VISUALIZATION VISU_Home  // 800x480
END_VISUALIZATION

(* stored: Version 1.1.0.1, ProductVersion 3.1.4026.18
   Visu VISU_Home: Id {d27000f4-d958-4452-9039-a62c97db2c5c} *)
